Universal Robots PolyScope program: ATI Simple Demo Program.urp

Program ATI Simple Demo Program (installation=default directory=/programs/usbdisk/20220721 createdIn=3.1.18024.0 lastSavedIn=3.15.6.106324 robotSerialNumber=2016353406)
Calibrated DH parameters: a=[0.000241, -0.156882, -0.391168, -0.000034, 0.000033, 0]; d=[0.08909, 1210.353649, -1202.089359, -8.154207, 0.094912, 0.082482]; alpha=[1.570962, 0.000326, -0.003342, 1.570446, -1.570439, 0]; deltaTheta=[0.000082, 1.192638, -1.263181, 0.0705, 0.00007, 0.000052]
BeforeStart
  Folder Move to Initial start position
    MoveJ speed 60 deg/s, acceleration 80 deg/s^2 (useActiveTCP=false)
      'CAUTION: check reachability or edit Waypoint before running Demo!'
      Waypoint Start: TCP in base x=-436.352 y=579.706 z=355.306 mm, rx=3.1399 ry=-0.0472 rz=-0.0056 rad; joints [-61.803, -57.175, 58.456, -91.289, 270.047, 29.954] deg
  URCap F/T Sensor Command (ATI Axia Force/Torque Sensor, ATI Industrial Automation) dataModel(WEIGHT=0.025, running=Enable)
  'Initialize variable for use in thread'
  ATI_FT_rawdata := ati_ftsensor.get_raw_ft()
Robot Program (runOnlyOnce=false)
  Folder Bias the sensor
    Wait Sleep waitTime=0.5
    URCap F/T Sensor Command (ATI Axia Force/Torque Sensor, ATI Industrial Automation) dataModel(running=Bias)
    Wait Sleep waitTime=0.5
  'This Demo program shows multiple ways to read F/T data for a "Force Search" in Z direction'
  Folder METHOD 1: Read F/T data via native UR command
    MoveL speed 40 mm/s, acceleration 200 mm/s^2 (useActiveTCP=false) feature=Base
      'Move down until the tool touches a surface'
      If force()<2 (checkContinuously=true)
        Waypoint RelativeMotionZ (Relative): relativeFromPosition TCP in base x=-99.537 y=-399.332 z=353.883 mm, rx=0.0027 ry=-3.1384 rz=-0.0008 rad; joints [-88.578, -78.615, -111.599, -79.821, 89.816, 1.322] deg; TCP in base x=-100.895 y=-399.448 z=-109.905 mm, rx=-0.0035 ry=-3.1383 rz=-0.0004 rad; joints [-88.578, -139.653, -133.528, 3.146, 89.816, 1.322] deg
      'Wait, then return to the start position'
      Wait Sleep waitTime=1
      Waypoint Start: TCP in base x=-436.352 y=579.706 z=355.306 mm, rx=3.1399 ry=-0.0472 rz=-0.0056 rad; joints [-61.803, -57.175, 58.456, -91.289, 270.047, 29.954] deg
  Folder METHOD 2: Read raw F/T data via ATI F/T URCap command
    MoveL speed 40 mm/s, acceleration 200 mm/s^2 (useActiveTCP=false) feature=Base
      'Move down until the tool touches a surface'
      If ATI_FT_Fz>-2 (checkContinuously=true)
        Waypoint RelativeMotionZ (Relative): relativeFromPosition TCP in base x=-99.537 y=-399.332 z=353.883 mm, rx=0.0027 ry=-3.1384 rz=-0.0008 rad; joints [-88.578, -78.615, -111.599, -79.821, 89.816, 1.322] deg; TCP in base x=-100.895 y=-399.448 z=-109.905 mm, rx=-0.0035 ry=-3.1383 rz=-0.0004 rad; joints [-88.578, -139.653, -133.528, 3.146, 89.816, 1.322] deg
      'Wait, then return to the start position'
      Wait Sleep waitTime=1
      Waypoint Start: TCP in base x=-436.352 y=579.706 z=355.306 mm, rx=3.1399 ry=-0.0472 rz=-0.0056 rad; joints [-61.803, -57.175, 58.456, -91.289, 270.047, 29.954] deg
Thread Thread_1 (runOnlyOnce=false)
  'MONITOR THIS DATA DURING PROGRAM FROM "Variables" TAB'
  Wait Sleep waitTime=0.01
  'Read sensor F/T Data using F/T URCap command, & assign it to a variable.'
  'This is the raw data directly from the sensor, in the sensor coordinate frame.'
  'With every loop of the thread, update the raw F/T data reading.'
  ATI_FT_rawdata := ati_ftsensor.get_raw_ft()
  'Fz is the 3rd element of the ATI_FT_data variable.'
  'NOTE: Pressing sensor in Z causes a -Z force (if no sensor Tool Transform applied)'
  ATI_FT_Fz := ATI_FT_rawdata[2]
  'F/T sensor data can also be read from native UR commands.'
  'Data read from UR commands will have transformations applied.'
  '(it is in robot base frame, not in the sensor coordinate frame).'
  ' UR Command get_tcp_force() gives TCP force in coordinate frame of robot base.'
  FTinBaseFrame := get_tcp_force()
  'UR command force() gives the Norm of get_tcp_force().'
  ForceNorm := force()
